(* PLC project mode, Dassault Systèmes ControlBuild 2024x *)
(* stored: creationDateTime 2023-10-03T11:13:41-01:00 *)

FUNCTION_BLOCK bottling_line.mode
  VAR_INPUT
    powerUpPB : BOOL := false;
    emergencyStopPB : BOOL := false;
    manual : BOOL := false;
    auto : BOOL := false;
  END_VAR
  VAR_INPUT
    acknowledgePB : BOOL := false;
  END_VAR
  VAR_OUTPUT
    powerUp : BOOL := false;
  END_VAR
  VAR_OUTPUT
    autoMode : BOOL := false;
    manualMode : BOOL := false;
  END_VAR
  VAR
    emStp : BOOL := false;
  END_VAR
  VAR  (* added by the conversion: wires and edge detectors of the diagram *)
    R_TRIG1 : R_TRIG;
    F_TRIG2 : F_TRIG;
  END_VAR

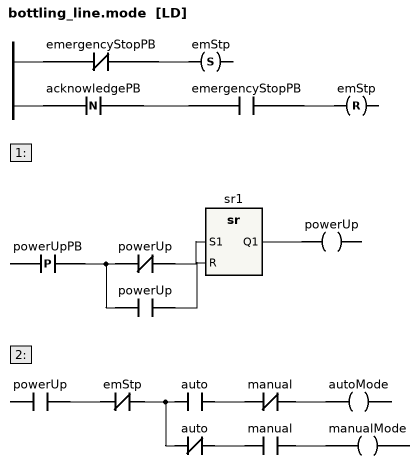
(* LD diagram, written out as Structured Text *)
1:
R_TRIG1(CLK := powerUpPB);
sr1(S1 := R_TRIG1.Q AND NOT powerUp, R := R_TRIG1.Q AND powerUp);
powerUp := sr1.Q1;
2:
IF NOT emergencyStopPB THEN emStp := TRUE; END_IF;
F_TRIG2(CLK := acknowledgePB);
IF F_TRIG2.Q AND emergencyStopPB THEN emStp := FALSE; END_IF;
autoMode := powerUp AND NOT emStp AND auto AND NOT manual;
manualMode := powerUp AND NOT emStp AND NOT auto AND manual;
END_FUNCTION_BLOCK
